// TwinCAT 3 PLC project CNM_OpModeHandlingInterfaces
// Title: CNM_OpModeHandlingInterfaces
// Company: ekvip automation GmbH
// Author: tsch
// ProjectVersion: 0.1.1.0
// Description: Providing interfaces that define handling operation modes in an industrial machine.
// ProgramVersion: 3.1.4026.19
// libraries:
//   CNM_AbstractObject, * (ekvip automation GmbH)
//   CNM_MessageInterfaces, * (ekvip automation GmbH)
//   CNM_ReturnTypes, * (ekvip automation GmbH)
//   Tc2_System, * (Beckhoff Automation GmbH)
// project tree:
//   Interfaces/Handler/ IOpModeHandlerMessageService.TcIO, INodeRequestProvider.TcIO, IOpModeHandler.TcIO, ISafetyReleaseDistributor.TcIO, ISafetySwitch.TcIO, IOpModeHandlerHmi.TcIO
//   Interfaces/Hmi/ IHmiApi.TcIO, IModeConditionProvider.TcIO
//   Interfaces/ IRunable.TcIO
//   Interfaces/Mode/ IModeBehaviour.TcIO, IModeProvider.TcIO, IModeSelect.TcIO
//   Interfaces/Node/Base/ INode.TcIO, INodeControl.TcIO, INodeRequest.TcIO
//   Interfaces/Node/ ICyclicNode.TcIO, INodeMessageService.TcIO
//   Interfaces/Node/OperationalNode/ IModeNode.TcIO, IOpModes.TcIO
//   Project Information/ F_GetCompany.TcPOU, F_GetTitle.TcPOU, F_GetVersion.TcPOU
//   Types/ ButtonStruct.TcDUT, HmiStates.TcDUT, ModeControlButtonStruct.TcDUT, NodeHandlerControlStruct.TcDUT
//   Version/ Global_Version.TcGVL

// ---- Types/ButtonStruct.TcDUT
TYPE ButtonStruct :
STRUCT
	text : Tc2_System.T_MaxString;
	enabled :BOOL := FALSE;
	visible :BOOL := FALSE;
	pressed :BOOL := FALSE;
END_STRUCT
END_TYPE

// ---- Types/HmiStates.TcDUT
{attribute 'qualified_only'}
{attribute 'strict'}
{attribute 'to_string'}
TYPE HmiStates :
(
	STOPPED := 0,
	HOME,
	RUNNING,
	PAUSE,
	STOP_PENDING,
	OFFLINE
);
END_TYPE

// ---- Types/ModeControlButtonStruct.TcDUT
TYPE ModeControlButtonStruct :
STRUCT
	Start :ButtonStruct:= (text:='%l%start%/l%');
	Stop :ButtonStruct:= (text:='%l%stop%/l%');
	StopRequest :ButtonStruct:= (text:='%l%stopRequest%/l%');
	StepMode :ButtonStruct:= (text:='%l%stepMode%/l%');
	Pause :ButtonStruct:= (text:='%l%pause%/l%');
END_STRUCT
END_TYPE

// ---- Types/NodeHandlerControlStruct.TcDUT
TYPE NodeHandlerControlStruct :
STRUCT
	stop :BOOL; // stop request for stop after end of cycle
	override :LREAL; // velocity orverride in % [0.0 ... 100.0]
END_STRUCT
END_TYPE

// ---- Version/Global_Version.TcGVL
{attribute 'TcGenerated'}
{attribute 'no-analysis'}
{attribute 'linkalways'}
// This function has been automatically generated from the project information.
VAR_GLOBAL CONSTANT
	{attribute 'const_non_replaced'}
	stLibVersion_CNM_OpModeHandlingInterfaces : ST_LibVersion := (iMajor := 0, iMinor := 1, iBuild := 1, iRevision := 0, nFlags := 0, sVersion := '0.1.1.0');
END_VAR

// ---- Interfaces/Handler/IOpModeHandlerMessageService.TcIO
(*
## short summary

This interface extends the IMessageInterface with the possibility to inject a global message service where the errors will be forwarded to.

legal notes
=================
| SPDX-FileCopyrightText: © 2024 ekvip automation GmbH <info@ekvip.de>
| SPDX-License-Identifier: Apache-2.0
| For details check: Apache-2.0_

.. _Apache-2.0: https://www.apache.org/licenses/LICENSE-2.0

.. </legal notes>  

*)

INTERFACE IOpModeHandlerMessageService EXTENDS CNM_MessageInterfaces.IMessageService

(*
## short summary

This property can be used to set the global message service interface during initialization.
The node message service will inform the node about the error and then forward the error to the global message service for handling the error.

legal notes
=================
| SPDX-FileCopyrightText: © 2025 ekvip automation GmbH <info@ekvip.de>
| SPDX-License-Identifier: Apache-2.0
| For details check: Apache-2.0_

.. _Apache-2.0: https://www.apache.org/licenses/LICENSE-2.0

.. </legal notes>  

*)

PROPERTY globalMessageService :CNM_MessageInterfaces.IMessageService
SET
END_SET
END_PROPERTY

END_INTERFACE

// ---- Interfaces/Handler/INodeRequestProvider.TcIO
(*
## short summary

This interface provides interfaces for the default node requests: disable, enable, initialize and stopImmediate.

legal notes
=================
| SPDX-FileCopyrightText: © 2024 ekvip automation GmbH <info@ekvip.de>
| SPDX-License-Identifier: Apache-2.0
| For details check: Apache-2.0_

.. _Apache-2.0: https://www.apache.org/licenses/LICENSE-2.0

.. </legal notes>  

*)

INTERFACE INodeRequestProvider EXTENDS __SYSTEM.IQueryInterface

(*
## short summary

This property returns the interface for the disabling request.

legal notes
=================
| SPDX-FileCopyrightText: © 2024 ekvip automation GmbH <info@ekvip.de>
| SPDX-License-Identifier: Apache-2.0
| For details check: Apache-2.0_

.. _Apache-2.0: https://www.apache.org/licenses/LICENSE-2.0

.. </legal notes>  

*)

PROPERTY disable :INodeRequest
GET
END_GET
END_PROPERTY

(*
## short summary

This property returns the interface for the disabling request.

legal notes
=================
| SPDX-FileCopyrightText: © 2024 ekvip automation GmbH <info@ekvip.de>
| SPDX-License-Identifier: Apache-2.0
| For details check: Apache-2.0_

.. _Apache-2.0: https://www.apache.org/licenses/LICENSE-2.0

.. </legal notes>  

*)

PROPERTY enable :INodeRequest
GET
END_GET
END_PROPERTY

(*
## short summary

This property returns the interface for the disabling request.

legal notes
=================
| SPDX-FileCopyrightText: © 2024 ekvip automation GmbH <info@ekvip.de>
| SPDX-License-Identifier: Apache-2.0
| For details check: Apache-2.0_

.. _Apache-2.0: https://www.apache.org/licenses/LICENSE-2.0

.. </legal notes>  

*)

PROPERTY initialize :INodeRequest
GET
END_GET
END_PROPERTY

(*
## short summary

This property returns the interface for the disabling request.

legal notes
=================
| SPDX-FileCopyrightText: © 2024 ekvip automation GmbH <info@ekvip.de>
| SPDX-License-Identifier: Apache-2.0
| For details check: Apache-2.0_

.. _Apache-2.0: https://www.apache.org/licenses/LICENSE-2.0

.. </legal notes>  

*)

PROPERTY stopImmediate :INodeRequest
GET
END_GET
END_PROPERTY

END_INTERFACE

// ---- Interfaces/Handler/IOpModeHandler.TcIO
(*
## short summary

This interface provides the cyclic run method and the fluent requests interface for a operation mode handler.

legal notes
=================
| SPDX-FileCopyrightText: © 2024 ekvip automation GmbH <info@ekvip.de>
| SPDX-License-Identifier: Apache-2.0
| For details check: Apache-2.0_

.. _Apache-2.0: https://www.apache.org/licenses/LICENSE-2.0

.. </legal notes>  

*)
INTERFACE IOpModeHandler EXTENDS CNM_AbstractObject.IObject, ISafetySwitch, IOpModeHandlerHmi, IRunable

END_INTERFACE

// ---- Interfaces/Handler/ISafetyReleaseDistributor.TcIO
(*
## short summary

This interface provides an subscription for a global safety release notification and should be implemented by the safety handler.

legal notes
=================
| SPDX-FileCopyrightText: © 2024 ekvip automation GmbH <info@ekvip.de>
| SPDX-License-Identifier: Apache-2.0
| For details check: Apache-2.0_

.. _Apache-2.0: https://www.apache.org/licenses/LICENSE-2.0

.. </legal notes>  

*)

INTERFACE ISafetyReleaseDistributor EXTENDS IRunable

(*
## short summary

This method adds the subscriber to a subscribption list. All subscribers are going to be notified, if the safety release changes.

legal notes
=================
| SPDX-FileCopyrightText: © 2022 ekvip automation GmbH <info@ekvip.de>
| SPDX-License-Identifier: Apache-2.0
| For details check: Apache-2.0_

.. _Apache-2.0: https://www.apache.org/licenses/LICENSE-2.0

.. </legal notes>  

*)

METHOD subscribe
VAR_INPUT
	(* class with the Interface ISafetySwitch, that can be switched on/off *)
	subscriber	:ISafetySwitch;
END_VAR
END_METHOD

END_INTERFACE

// ---- Interfaces/Handler/ISafetySwitch.TcIO
(*
## short summary

This interface needs to be implemented for a subscription to the ISafetyReleaseDistributer interface.
The provided methods switchOn and switchOff are automatically called if the safety release changes.

legal notes
=================
| SPDX-FileCopyrightText: © 2024 ekvip automation GmbH <info@ekvip.de>
| SPDX-License-Identifier: Apache-2.0
| For details check: Apache-2.0_

.. _Apache-2.0: https://www.apache.org/licenses/LICENSE-2.0

.. </legal notes>  

*)

INTERFACE ISafetySwitch EXTENDS CNM_AbstractObject.IObject

(*
## short summary

This property indicates that the unit is enabled and all safety requirements are met.

legal notes
=================
| SPDX-FileCopyrightText: © 2024 ekvip automation GmbH <info@ekvip.de>
| SPDX-License-Identifier: Apache-2.0
| For details check: Apache-2.0_

.. _Apache-2.0: https://www.apache.org/licenses/LICENSE-2.0

.. </legal notes>  

*)
PROPERTY isSwitchedOn : BOOL
GET
END_GET
END_PROPERTY

(*
## short summary

This method disables the unit if not all safety requirements are met. It Should be called only from the safety management.

legal notes
=================
| SPDX-FileCopyrightText: © 2024 ekvip automation GmbH <info@ekvip.de>
| SPDX-License-Identifier: Apache-2.0
| For details check: Apache-2.0_

.. _Apache-2.0: https://www.apache.org/licenses/LICENSE-2.0

.. </legal notes>  

*)

METHOD switchOff
END_METHOD

(*
## short summary

This method enables the unit if all safety requirements are met. It Should be called only from the safety management.

legal notes
=================
| SPDX-FileCopyrightText: © 2024 ekvip automation GmbH <info@ekvip.de>
| SPDX-License-Identifier: Apache-2.0
| For details check: Apache-2.0_

.. _Apache-2.0: https://www.apache.org/licenses/LICENSE-2.0

.. </legal notes>  

*)

METHOD switchOn
END_METHOD

END_INTERFACE

// ---- Interfaces/Handler/IOpModeHandlerHmi.TcIO
(*
## short summary
This interface provides an API to control the operation mode handler.

legal notes
=================
| SPDX-FileCopyrightText: © 2024 ekvip automation GmbH <info@ekvip.de>
| SPDX-License-Identifier: Apache-2.0
| For details check: Apache-2.0_

.. _Apache-2.0: https://www.apache.org/licenses/LICENSE-2.0

.. </legal notes>  

*)
INTERFACE IOpModeHandlerHmi EXTENDS CNM_AbstractObject.IObject

(*
## short summary
This methods enables the stepping operation on a given node and all of its subnodes.

legal notes
=================
| SPDX-FileCopyrightText: © 2025 ekvip automation GmbH <info@ekvip.de>
| SPDX-License-Identifier: Apache-2.0
| For details check: Apache-2.0_

.. _Apache-2.0: https://www.apache.org/licenses/LICENSE-2.0

.. </legal notes>  

*)

METHOD enableStepping : CNM_ReturnTypes.SingleExecutionResult
VAR_INPUT
	(* the node on which stepping should be enabled *)
	node :INode;
END_VAR
END_METHOD

(*
## short summary
This property can be used to inject a message service. Messages will be forwarded to that message service if it is set.

legal notes
=================
| SPDX-FileCopyrightText: © 2025 ekvip automation GmbH <info@ekvip.de>
| SPDX-License-Identifier: Apache-2.0
| For details check: Apache-2.0_

.. _Apache-2.0: https://www.apache.org/licenses/LICENSE-2.0

.. </legal notes>  

*)

PROPERTY globalMessageService : CNM_MessageInterfaces.IMessageService
SET
END_SET
END_PROPERTY

(*
## short summary
This property can be used to set the global override from the HMI and to read back the current override for the HMI.

**information**: the override has a range from 0.0 to 100.0 and will be limited to the upper/lower bound.

legal notes
=================
| SPDX-FileCopyrightText: © 2024 ekvip automation GmbH <info@ekvip.de>
| SPDX-License-Identifier: Apache-2.0
| For details check: Apache-2.0_

.. _Apache-2.0: https://www.apache.org/licenses/LICENSE-2.0

.. </legal notes>  

*)

PROPERTY globalOverride : LREAL
GET
END_GET
SET
END_SET
END_PROPERTY

(*
## short summary
This property indicates that a operation is being executed.

legal notes
=================
| SPDX-FileCopyrightText: © 2025 ekvip automation GmbH <info@ekvip.de>
| SPDX-License-Identifier: Apache-2.0
| For details check: Apache-2.0_

.. _Apache-2.0: https://www.apache.org/licenses/LICENSE-2.0

.. </legal notes>  

*)

PROPERTY modeIsExecuting : BOOL
GET
END_GET
END_PROPERTY

(*
## short summary
This property can be used to pause the currently running operation mode from the HMI and to read back if the mode is paused.

legal notes
=================
| SPDX-FileCopyrightText: © 2024 ekvip automation GmbH <info@ekvip.de>
| SPDX-License-Identifier: Apache-2.0
| For details check: Apache-2.0_

.. _Apache-2.0: https://www.apache.org/licenses/LICENSE-2.0

.. </legal notes>  

*)

PROPERTY pause : BOOL
GET
END_GET
SET
END_SET
END_PROPERTY

(*
## short summary
This property returns the INodeHmiApi interface of the root node from this opmode handler.

legal notes
=================
| SPDX-FileCopyrightText: © 2024 ekvip automation GmbH <info@ekvip.de>
| SPDX-License-Identifier: Apache-2.0
| For details check: Apache-2.0_

.. _Apache-2.0: https://www.apache.org/licenses/LICENSE-2.0

.. </legal notes>  

*)

PROPERTY rootNode :INode
GET
END_GET
END_PROPERTY

(*
## short summary
This method sets a mode for the rootnode or, if specified, for a single node and its subnodes.
It is only allowed to overwrite the mode if the rootNode or the specified node is not in busy state.

legal notes
=================
| SPDX-FileCopyrightText: © 2024 ekvip automation GmbH <info@ekvip.de>
| SPDX-License-Identifier: Apache-2.0
| For details check: Apache-2.0_

.. _Apache-2.0: https://www.apache.org/licenses/LICENSE-2.0

.. </legal notes>  

## example
set it for the whole machine:
```
myOpmodeHandler.setMode(
	mode := automaticMode
);
```

overwrite the mode of specified node:
```
myOpmodeHandler.setMode(
	mode := serviceMode,
	node := despensingUnit
);
```

*)
METHOD setMode : CNM_ReturnTypes.SingleExecutionResult
VAR_INPUT
	(* the mode instance that should be set *)
	mode : IModeBehaviour;
	(* optionally: a specified node in the tree that is not the subtree (if 0, the rootNode will be adressed) *)
	node : IModeNode := 0;
END_VAR
END_METHOD

(*
## short summary
This method starts the currently selected operation mode if all safety requirements are met.

legal notes
=================
| SPDX-FileCopyrightText: © 2024 ekvip automation GmbH <info@ekvip.de>
| SPDX-License-Identifier: Apache-2.0
| For details check: Apache-2.0_

.. _Apache-2.0: https://www.apache.org/licenses/LICENSE-2.0

.. </legal notes>  

## example
```
CASE step OF
	0:	// choose and set mode
		IF (handler.setMode(automaticMode) = SUCCESS ) THEN
			step := 1;
		END_IF
	1:	// start mode
		IF (handler.startMode() = SUCCESS) THEN
			step := 2;
		END_IF
	2: // stop mode if requested
		IF ( stopRequested ) THEN
			IF ( handler.stopMode() = SUCCESS ) THEN
				step := 0;
			END_IF
		END_IF
END_CASE
```

*)

METHOD startMode :CNM_ReturnTypes.SingleExecutionResult
VAR_INPUT
	(* optionally: a specified node in the tree that is not the subtree (if 0, the rootNode will be adressed) *)
	node : INode := 0;
END_VAR
END_METHOD

(*
## short summary
This method stops the currently running operation mode.
If the immediately flag is set, the current operation modewill be aborted and the machine will execute a fast stop.
If it is not set, the stop request flag for all nodes will be set and the operation modes should exit with a defined state.

legal notes
=================
| SPDX-FileCopyrightText: © 2024 ekvip automation GmbH <info@ekvip.de>
| SPDX-License-Identifier: Apache-2.0
| For details check: Apache-2.0_

.. _Apache-2.0: https://www.apache.org/licenses/LICENSE-2.0

.. </legal notes>  

## parameters
**return**: `CNM_ReturnTypes.SingleExecutionState`
- `SUCCESS`: the mode was stopped
- `BUSY`: mode is still stopping

## example
```
CASE step OF
	0:	// choose and set mode
		IF (handler.setMode(automaticMode) = SUCCESS ) THEN
			step := 1;
		END_IF
	1:	// start mode
		IF (handler.startMode() = SUCCESS) THEN
			step := 2;
		END_IF
	2: // stop mode if requested
		IF ( stopRequested ) THEN
			IF ( handler.stopMode() = SUCCESS ) THEN
				step := 0;
			END_IF
		END_IF
END_CASE
```

*)

METHOD stopMode : CNM_ReturnTypes.SingleExecutionState
VAR_INPUT
	(* if this flag is set, the current operation mode will be aborted and the machine will execute a fast stop *)
	immediately :BOOL := FALSE;
END_VAR
END_METHOD

END_INTERFACE

// ---- Interfaces/Hmi/IHmiApi.TcIO
(*
## short summary

This interface provides control methods and properties for a HMI handler class that are called by the CNM HMI framework.

legal notes
=================
| SPDX-FileCopyrightText: © 2024 ekvip automation GmbH <info@ekvip.de>
| SPDX-License-Identifier: Apache-2.0
| For details check: Apache-2.0_

.. _Apache-2.0: https://www.apache.org/licenses/LICENSE-2.0

.. </legal notes>  

*)

INTERFACE IHmiApi EXTENDS __SYSTEM.IQueryInterface, IRunable

(*
## short summary

This method returns the instance path of the root node of the operation mode handler.
It is used for the HMI tree building mechanism.

legal notes
=================
| SPDX-FileCopyrightText: © 2024 ekvip automation GmbH <info@ekvip.de>
| SPDX-License-Identifier: Apache-2.0
| For details check: Apache-2.0_

.. _Apache-2.0: https://www.apache.org/licenses/LICENSE-2.0

.. </legal notes>  

*)

{attribute 'TcRpcEnable'}
METHOD getRootNodeName : Tc2_System.T_MaxString
END_METHOD

(*
## short summary

This property is true if the operation mode handler has a safety release.

legal notes
=================
| SPDX-FileCopyrightText: © 2024 ekvip automation GmbH <info@ekvip.de>
| SPDX-License-Identifier: Apache-2.0
| For details check: Apache-2.0_

.. _Apache-2.0: https://www.apache.org/licenses/LICENSE-2.0

.. </legal notes>  

*)

{attribute 'monitoring':='call'}
PROPERTY IsSafetyOk : BOOL
GET
END_GET
END_PROPERTY

(*
## short summary

This property can returns the root node state for currently active operation mode.

legal notes
=================
| SPDX-FileCopyrightText: © 2024 ekvip automation GmbH <info@ekvip.de>
| SPDX-License-Identifier: Apache-2.0
| For details check: Apache-2.0_

.. _Apache-2.0: https://www.apache.org/licenses/LICENSE-2.0

.. </legal notes>  

*)

{attribute 'monitoring' := 'call'}
PROPERTY OpModeState : CNM_ReturnTypes.SingleExecutionState
GET
END_GET
END_PROPERTY

(*
## short summary

This property can be used to pause the currently running operation mode from the HMI and to read back if the mode is paused.

legal notes
=================
| SPDX-FileCopyrightText: © 2024 ekvip automation GmbH <info@ekvip.de>
| SPDX-License-Identifier: Apache-2.0
| For details check: Apache-2.0_

.. _Apache-2.0: https://www.apache.org/licenses/LICENSE-2.0

.. </legal notes>  

*)

{attribute 'monitoring':='call'}
PROPERTY pause : BOOL
GET
END_GET
SET
END_SET
END_PROPERTY

(*
## short summary

This property shows that the root node (and so the whole machine) is waiting for a step signal when step mode is enabled.

legal notes
=================
| SPDX-FileCopyrightText: © 2024 ekvip automation GmbH <info@ekvip.de>
| SPDX-License-Identifier: Apache-2.0
| For details check: Apache-2.0_

.. _Apache-2.0: https://www.apache.org/licenses/LICENSE-2.0

.. </legal notes>  

*)

{attribute 'monitoring' := 'call'}
PROPERTY rootNodeWaitingForStep : BOOL
GET
END_GET
END_PROPERTY

(*
## short summary

This property setter sends the step signal to all nodes of the machine.
If the step mode is enabled, the step signal will be set for exactly one PLC cycle.
If the step mode isn't enabled, the step signal won't have any effect at all.

legal notes
=================
| SPDX-FileCopyrightText: © 2024 ekvip automation GmbH <info@ekvip.de>
| SPDX-License-Identifier: Apache-2.0
| For details check: Apache-2.0_

.. _Apache-2.0: https://www.apache.org/licenses/LICENSE-2.0

.. </legal notes>  

*)

{attribute 'monitoring':='call'}
PROPERTY step : BOOL
SET
END_SET
END_PROPERTY

END_INTERFACE

// ---- Interfaces/Hmi/IModeConditionProvider.TcIO
(*
## short summary

This interface provides a method that checks for each mode if it can be started.

legal notes
=================
| SPDX-FileCopyrightText: © 2024 ekvip automation GmbH <info@ekvip.de>
| SPDX-License-Identifier: Apache-2.0
| For details check: Apache-2.0_

.. _Apache-2.0: https://www.apache.org/licenses/LICENSE-2.0

.. </legal notes>  

*)

INTERFACE IModeConditionProvider

(*
## short summary

This method checks the start conditions for the selected operation mode.
If the mode is allowed to be started, it returns TRUE.

legal notes
=================
| SPDX-FileCopyrightText: © 2024 ekvip automation GmbH <info@ekvip.de>
| SPDX-License-Identifier: Apache-2.0
| For details check: Apache-2.0_

.. _Apache-2.0: https://www.apache.org/licenses/LICENSE-2.0

.. </legal notes>  

*)

METHOD checkModeIsAllowed : BOOL
VAR_INPUT
	mode :UDINT;
	node :INode;
END_VAR
END_METHOD

END_INTERFACE

// ---- Interfaces/IRunable.TcIO
(*
## short summary

This interface provides a void run() method without parameters.

legal notes
=================
| SPDX-FileCopyrightText: © 2025 ekvip automation GmbH <info@ekvip.de>
| SPDX-License-Identifier: Apache-2.0
| For details check: Apache-2.0_

.. _Apache-2.0: https://www.apache.org/licenses/LICENSE-2.0

.. </legal notes>  

*)

INTERFACE IRunable EXTENDS CNM_AbstractObject.IObject

(*
## short summary

A method that should be called cyclically to update and execute a class instance.

legal notes
=================
| SPDX-FileCopyrightText: © 2025 ekvip automation GmbH <info@ekvip.de>
| SPDX-License-Identifier: Apache-2.0
| For details check: Apache-2.0_

.. _Apache-2.0: https://www.apache.org/licenses/LICENSE-2.0

.. </legal notes>  

*)

METHOD run
END_METHOD

END_INTERFACE

// ---- Interfaces/Mode/IModeBehaviour.TcIO
(*
## short summary

This interface defines the methods needed for the mode delegates.

legal notes
=================
| SPDX-FileCopyrightText: © 2024 ekvip automation GmbH <info@ekvip.de>
| SPDX-License-Identifier: Apache-2.0
| For details check: Apache-2.0_

.. _Apache-2.0: https://www.apache.org/licenses/LICENSE-2.0

.. </legal notes>  

*)

INTERFACE IModeBehaviour EXTENDS CNM_AbstractObject.IObject

(*
## short summary

This property is intended to inform cyclic nodes (devices) that manual commands are allowed to be executed.
Usually only the manual mode behaviour sets this to true, but it may be also used for other custom modes if needed.

legal notes
=================
| SPDX-FileCopyrightText: © 2024 ekvip automation GmbH <info@ekvip.de>
| SPDX-License-Identifier: Apache-2.0
| For details check: Apache-2.0_

.. _Apache-2.0: https://www.apache.org/licenses/LICENSE-2.0

.. </legal notes>  

*)

PROPERTY enableManCmds : BOOL
GET
END_GET
END_PROPERTY

(*
## short summary

This method is called once for every node when a new oepration mode is started.
It is intended to inform the node that a new mode is startet, so you can throw events / MES notifications /  do data management here.

legal notes
=================
| SPDX-FileCopyrightText: © 2024 ekvip automation GmbH <info@ekvip.de>
| SPDX-License-Identifier: Apache-2.0
| For details check: Apache-2.0_

.. _Apache-2.0: https://www.apache.org/licenses/LICENSE-2.0

.. </legal notes>  

*)

METHOD enterMode
VAR_INPUT
	node : IOpModes;
END_VAR
END_METHOD

(*
## short summary

This method is called once for every node when the current operation mode is stopped.
It is intended to inform the node that the mode is stopped, so you can throw events / MES notifications /  do data management here.

legal notes
=================
| SPDX-FileCopyrightText: © 2024 ekvip automation GmbH <info@ekvip.de>
| SPDX-License-Identifier: Apache-2.0
| For details check: Apache-2.0_

.. _Apache-2.0: https://www.apache.org/licenses/LICENSE-2.0

.. </legal notes>  

*)

METHOD exitMode
VAR_INPUT
	node : IOpModes;
END_VAR
END_METHOD

(*
## short summary

This property returns the id that was used to request the mode delegate.
The mode provider class has to set it.

legal notes
=================
| SPDX-FileCopyrightText: © 2024 ekvip automation GmbH <info@ekvip.de>
| SPDX-License-Identifier: Apache-2.0
| For details check: Apache-2.0_

.. _Apache-2.0: https://www.apache.org/licenses/LICENSE-2.0

.. </legal notes>  

*)

PROPERTY id : UDINT
GET
END_GET
SET
END_SET
END_PROPERTY

(*
## short summary

This method is calling the operation mode methods for every node depending on the current behaviour.

legal notes
=================
| SPDX-FileCopyrightText: © 2024 ekvip automation GmbH <info@ekvip.de>
| SPDX-License-Identifier: Apache-2.0
| For details check: Apache-2.0_

.. _Apache-2.0: https://www.apache.org/licenses/LICENSE-2.0

.. </legal notes>  

*)

METHOD run :CNM_ReturnTypes.SingleExecutionState
VAR_INPUT
	execute :BOOL;
	pause :BOOL;
	node :IOpModes;
END_VAR
END_METHOD

END_INTERFACE

// ---- Interfaces/Mode/IModeProvider.TcIO
(*
## short summary

This interface defines method for a mode behaviour provider. 
It can be used to inject custom modes into the HMI class.  

legal notes
=================
| SPDX-FileCopyrightText: © 2024 ekvip automation GmbH <info@ekvip.de>
| SPDX-License-Identifier: Apache-2.0
| For details check: Apache-2.0_

.. _Apache-2.0: https://www.apache.org/licenses/LICENSE-2.0

.. </legal notes>  

*)

INTERFACE IModeProvider EXTENDS CNM_AbstractObject.IObject

(*
## short summary

A method that returns an interface to an instance of a mode behaviour.
It can be used to trabnslate the operation mode enum to a mode delegate. Overwrite this method for custom modes.

legal notes
=================
| SPDX-FileCopyrightText: © 2024 ekvip automation GmbH <info@ekvip.de>
| SPDX-License-Identifier: Apache-2.0
| For details check: Apache-2.0_

.. _Apache-2.0: https://www.apache.org/licenses/LICENSE-2.0

.. </legal notes>  

*)

METHOD getMode : IModeBehaviour
VAR_INPUT
	mode :UDINT;
END_VAR
END_METHOD

(*
## short summary

This property returns an IModeSelect that offers properties for the mandatory modes.
The modes are accessable via fluent interface, e.g. myModeFactory.mode.automaticMode.

legal notes
=================
| SPDX-FileCopyrightText: © 2024 ekvip automation GmbH <info@ekvip.de>
| SPDX-License-Identifier: Apache-2.0
| For details check: Apache-2.0_

.. _Apache-2.0: https://www.apache.org/licenses/LICENSE-2.0

.. </legal notes>  

*)

PROPERTY mode : IModeSelect
GET
END_GET
END_PROPERTY

END_INTERFACE

// ---- Interfaces/Mode/IModeSelect.TcIO
(*
## short summary

This is an interface to fluently provide the mandatory mode behaviours.

legal notes
=================
| SPDX-FileCopyrightText: © 2024 ekvip automation GmbH <info@ekvip.de>
| SPDX-License-Identifier: Apache-2.0
| For details check: Apache-2.0_

.. _Apache-2.0: https://www.apache.org/licenses/LICENSE-2.0

.. </legal notes>  

*)

INTERFACE IModeSelect EXTENDS CNM_AbstractObject.IObject

(*
## short summary

This property returns an IModeBehaviour that implements the delegate for the automatic mode.

legal notes
=================
| SPDX-FileCopyrightText: © 2024 ekvip automation GmbH <info@ekvip.de>
| SPDX-License-Identifier: Apache-2.0
| For details check: Apache-2.0_

.. _Apache-2.0: https://www.apache.org/licenses/LICENSE-2.0

.. </legal notes>  

*)
PROPERTY automaticMode : IModeBehaviour
GET
END_GET
END_PROPERTY

(*
## short summary

This property returns an IModeBehaviour that implements the delegate for the homing mode.

legal notes
=================
| SPDX-FileCopyrightText: © 2024 ekvip automation GmbH <info@ekvip.de>
| SPDX-License-Identifier: Apache-2.0
| For details check: Apache-2.0_

.. _Apache-2.0: https://www.apache.org/licenses/LICENSE-2.0

.. </legal notes>  

*)

PROPERTY homingMode : IModeBehaviour
GET
END_GET
END_PROPERTY

(*
## short summary

This property returns an IModeBehaviour that implements the delegate for the manual mode.

legal notes
=================
| SPDX-FileCopyrightText: © 2024 ekvip automation GmbH <info@ekvip.de>
| SPDX-License-Identifier: Apache-2.0
| For details check: Apache-2.0_

.. _Apache-2.0: https://www.apache.org/licenses/LICENSE-2.0

.. </legal notes>  

*)

PROPERTY manualMode : IModeBehaviour
GET
END_GET
END_PROPERTY

(*
## short summary

This property returns an IModeBehaviour that implements the delegate for no operation mode.

legal notes
=================
| SPDX-FileCopyrightText: © 2025 ekvip automation GmbH <info@ekvip.de>
| SPDX-License-Identifier: Apache-2.0
| For details check: Apache-2.0_

.. _Apache-2.0: https://www.apache.org/licenses/LICENSE-2.0

.. </legal notes>  

*)

PROPERTY noMode : IModeBehaviour
GET
END_GET
END_PROPERTY

END_INTERFACE

// ---- Interfaces/Node/Base/INode.TcIO
(*
## short summary
This interface provides methods and properties that every node needs to implement.
Some of the methods and properties are used for the CNM HMI framework.

legal notes
=================
| SPDX-FileCopyrightText: © 2024 ekvip automation GmbH <info@ekvip.de>
| SPDX-License-Identifier: Apache-2.0
| For details check: Apache-2.0_

.. _Apache-2.0: https://www.apache.org/licenses/LICENSE-2.0

.. </legal notes>  

*)

INTERFACE INode EXTENDS CNM_AbstractObject.IObject

(*
## short summary
This property returns the id of the mode that is currently propagated.
It reflects the hmi selection.

legal notes
=================
| SPDX-FileCopyrightText: © 2024 ekvip automation GmbH <info@ekvip.de>
| SPDX-License-Identifier: Apache-2.0
| For details check: Apache-2.0_

.. _Apache-2.0: https://www.apache.org/licenses/LICENSE-2.0

.. </legal notes>  

*)

PROPERTY currentModeId : UDINT
GET
END_GET
END_PROPERTY

(*
## short summary
This method disables a node (E.g. axes should be disabled). It can take mutliple cycles. It has to be implemented for every node/device.
The execute input needs a rising edge to execute the method.
If there is nothing to disable, just return a 'SUCCESS' state.

This method is called automatically by the operation mode handler.

legal notes
=================
| SPDX-FileCopyrightText: © 2024 ekvip automation GmbH <info@ekvip.de>
| SPDX-License-Identifier: Apache-2.0
| For details check: Apache-2.0_

.. _Apache-2.0: https://www.apache.org/licenses/LICENSE-2.0

.. </legal notes>  

*)

METHOD disable : CNM_ReturnTypes.SingleExecutionState
VAR_INPUT
	execute :BOOL;
END_VAR
END_METHOD

(*
## short summary
This method enables a node. It can take mutliple cycles. It has to be implemented for every node/device.
The intention is to enable devices here, e.g. axes, laser, dispenser etc.
The execute input needs a rising edge to execute the method.
If there is nothing to enable, just return a 'SUCCESS' state.

This method is called automatically by the operation mode handler.

legal notes
=================
| SPDX-FileCopyrightText: © 2024 ekvip automation GmbH <info@ekvip.de>
| SPDX-License-Identifier: Apache-2.0
| For details check: Apache-2.0_

.. _Apache-2.0: https://www.apache.org/licenses/LICENSE-2.0

.. </legal notes>  

*)
METHOD enable : CNM_ReturnTypes.SingleExecutionState
VAR_INPUT
	execute :BOOL;
END_VAR
END_METHOD

(*
## short summary
This property is used to enable/disable manual stepping.

legal notes
=================
| SPDX-FileCopyrightText: © 2025 ekvip automation GmbH <info@ekvip.de>
| SPDX-License-Identifier: Apache-2.0
| For details check: Apache-2.0_

.. _Apache-2.0: https://www.apache.org/licenses/LICENSE-2.0

.. </legal notes>  

*)

PROPERTY enableStepping : BOOL
GET
END_GET
SET
END_SET
END_PROPERTY

(*
## short summary
This method returns the variable name for a subnode at a given array index of the internal array list.
It is required for the HMI connection to construct the node tree from the PLC on HMI side.
It is also intended to be called from the HMI via remote procedure call.

legal notes
=================
| SPDX-FileCopyrightText: © 2024 ekvip automation GmbH <info@ekvip.de>
| SPDX-License-Identifier: Apache-2.0
| For details check: Apache-2.0_

.. _Apache-2.0: https://www.apache.org/licenses/LICENSE-2.0

.. </legal notes>  

*)

METHOD getSubnodeName : CNM_AbstractObject.ObjectName
VAR_INPUT
	(*  index of a subnode in the subnode array list *)
	index :UDINT;
END_VAR
END_METHOD

(*
## short summary
This property indicates whether a node has an error. It is used by the CNM HMI.

legal notes
=================
| SPDX-FileCopyrightText: © 2024 ekvip automation GmbH <info@ekvip.de>
| SPDX-License-Identifier: Apache-2.0
| For details check: Apache-2.0_

.. _Apache-2.0: https://www.apache.org/licenses/LICENSE-2.0

.. </legal notes>  

*)
{attribute 'monitoring' := 'call'}
PROPERTY hasError : BOOL
GET
END_GET
SET
END_SET
END_PROPERTY

(*
## short summary
This method contains instructions and sequences for the init mode.
This mode is intended for initializing a machine, e.g. set references and parameters, establish a connection to global production systems (MES).
If the node should do nothing, return a 'SUCCESS'.
It should run until all initializations are done or the mode is stopped immedtiately or a stop request is raised.
This method is called automatically by the operation mode handler after PLC startup.

legal notes
=================
| SPDX-FileCopyrightText: © 2024 ekvip automation GmbH <info@ekvip.de>
| SPDX-License-Identifier: Apache-2.0
| For details check: Apache-2.0_

.. _Apache-2.0: https://www.apache.org/licenses/LICENSE-2.0

.. </legal notes>  

*)
METHOD initialize : CNM_ReturnTypes.SingleExecutionState
VAR_INPUT
	execute :BOOL;
END_VAR
END_METHOD

(*
## short summary
This property indicates that a node or subunit is home position. The getter evaluates the home property of all child nodes.  
It is used by the CNM HMI.

legal notes
=================
| SPDX-FileCopyrightText: © 2024 ekvip automation GmbH <info@ekvip.de>
| SPDX-License-Identifier: Apache-2.0
| For details check: Apache-2.0_

.. _Apache-2.0: https://www.apache.org/licenses/LICENSE-2.0

.. </legal notes>  

*)
{attribute 'monitoring' := 'call'}
PROPERTY isInHome : BOOL
GET
END_GET
SET
END_SET
END_PROPERTY

(*
## short summary
This property indicates that a node or subunit is waiting for a step signal. It is used by the CNM HMI.

legal notes
=================
| SPDX-FileCopyrightText: © 2024 ekvip automation GmbH <info@ekvip.de>
| SPDX-License-Identifier: Apache-2.0
| For details check: Apache-2.0_

.. _Apache-2.0: https://www.apache.org/licenses/LICENSE-2.0

.. </legal notes>  

*)
{attribute 'monitoring' := 'call'}
PROPERTY isWaitingForStep : BOOL
GET
END_GET
SET
END_SET
END_PROPERTY

(*
## short summary
This property is used to set a local override for single node. 
The local override will be multiplied with the global override.

legal notes
=================
| SPDX-FileCopyrightText: © 2024 ekvip automation GmbH <info@ekvip.de>
| SPDX-License-Identifier: Apache-2.0
| For details check: Apache-2.0_

.. _Apache-2.0: https://www.apache.org/licenses/LICENSE-2.0

.. </legal notes>  

*)
{attribute 'monitoring' := 'variable'}
PROPERTY localOverride : LREAL
GET
END_GET
SET
END_SET
END_PROPERTY

(*
## short summary
This property returns the interface to the instance mode data dto.

legal notes
=================
| SPDX-FileCopyrightText: © 2024 ekvip automation GmbH <info@ekvip.de>
| SPDX-License-Identifier: Apache-2.0
| For details check: Apache-2.0_

.. _Apache-2.0: https://www.apache.org/licenses/LICENSE-2.0

.. </legal notes>  

*)
PROPERTY nodeControl : INodeControl
GET
END_GET
END_PROPERTY

(*
## short summary
This property returns the state of the node for the current node request.
The unit is still running if the state is ''BUSY''.

legal notes
=================
| SPDX-FileCopyrightText: © 2024 ekvip automation GmbH <info@ekvip.de>
| SPDX-License-Identifier: Apache-2.0
| For details check: Apache-2.0_

.. _Apache-2.0: https://www.apache.org/licenses/LICENSE-2.0

.. </legal notes>  

*)
{attribute 'monitoring' := 'call'}
PROPERTY nodeState : CNM_ReturnTypes.SingleExecutionState
GET
END_GET
END_PROPERTY

(*
## short summary
This boolean can be used to set the step signal for a node for one plc cycle.

legal notes
=================
| SPDX-FileCopyrightText: © 2025 ekvip automation GmbH <info@ekvip.de>
| SPDX-License-Identifier: Apache-2.0
| For details check: Apache-2.0_

.. _Apache-2.0: https://www.apache.org/licenses/LICENSE-2.0

.. </legal notes>  

*)

PROPERTY step : BOOL
GET
END_GET
SET
END_SET
END_PROPERTY

(*
## short summary
This method executes stops all movements of a node. It has to be overwritten for every node.
E.g. axes should perform a quickstop, cylinders should be turned off, etc.
If the node should do nothing, return a 'SUCCESS'.
It should stop axes/cylinders/process (e.g. laser welding, dispensing) endless until the manual mode is stopped via stop request or immediate stop.
This method is called automatically by the operation mode handler before disabling the machine or if the operator selects an immediate stop.

**attention**: If this method returns the state 'ERROR', the operation mode handler automatically disables the whole machine!

legal notes
=================
| SPDX-FileCopyrightText: © 2024 ekvip automation GmbH <info@ekvip.de>
| SPDX-License-Identifier: Apache-2.0
| For details check: Apache-2.0_

.. _Apache-2.0: https://www.apache.org/licenses/LICENSE-2.0

.. </legal notes>  

*)

METHOD stopImmediate : CNM_ReturnTypes.SingleExecutionState
VAR_INPUT
	execute :BOOL;
END_VAR
END_METHOD

END_INTERFACE

// ---- Interfaces/Node/Base/INodeControl.TcIO
(*
## short summary

This interface provides a fluent way to access the global control signals (stopRequests, overrides, step requests).

legal notes
=================
| SPDX-FileCopyrightText: © 2024 ekvip automation GmbH <info@ekvip.de>
| SPDX-License-Identifier: Apache-2.0
| For details check: Apache-2.0_

.. _Apache-2.0: https://www.apache.org/licenses/LICENSE-2.0

.. </legal notes>  

*)
INTERFACE INodeControl EXTENDS __SYSTEM.IQueryInterface

(*
## short summary

This property returns the effective override for a node, which is the result of the multiplication of global and local override.

legal notes
=================
| SPDX-FileCopyrightText: © 2024 ekvip automation GmbH <info@ekvip.de>
| SPDX-License-Identifier: Apache-2.0
| For details check: Apache-2.0_

.. _Apache-2.0: https://www.apache.org/licenses/LICENSE-2.0

.. </legal notes>  

*)
PROPERTY override : LREAL
GET
END_GET
END_PROPERTY

(*
## short summary

This property represents the stop request signal which either the operator triggers from the HMI or which is set by an error.

legal notes
=================
| SPDX-FileCopyrightText: © 2024 ekvip automation GmbH <info@ekvip.de>
| SPDX-License-Identifier: Apache-2.0
| For details check: Apache-2.0_

.. _Apache-2.0: https://www.apache.org/licenses/LICENSE-2.0

.. </legal notes>  

*)
PROPERTY stopRequest : BOOL
GET
END_GET
END_PROPERTY

END_INTERFACE

// ---- Interfaces/Node/Base/INodeRequest.TcIO
(*
## short summary

This interface defines the methods needed for the node request delegates.

legal notes
=================
| SPDX-FileCopyrightText: © 2024 ekvip automation GmbH <info@ekvip.de>
| SPDX-License-Identifier: Apache-2.0
| For details check: Apache-2.0_

.. _Apache-2.0: https://www.apache.org/licenses/LICENSE-2.0

.. </legal notes>  

*)

INTERFACE INodeRequest EXTENDS __SYSTEM.IQueryInterface

(*
## short summary

This method is calling the node request methods for every node depending on the current request.

legal notes
=================
| SPDX-FileCopyrightText: © 2024 ekvip automation GmbH <info@ekvip.de>
| SPDX-License-Identifier: Apache-2.0
| For details check: Apache-2.0_

.. _Apache-2.0: https://www.apache.org/licenses/LICENSE-2.0

.. </legal notes>  

*)

METHOD run :CNM_ReturnTypes.SingleExecutionState
VAR_INPUT
	execute :BOOL;
	node :INode;
END_VAR
END_METHOD

END_INTERFACE

// ---- Interfaces/Node/ICyclicNode.TcIO
(*
## short summary

This interface extends the INode interface with a run method for a cyclically update/monitoring.
Examples for cyclic nodes are device drivers, meausurements or communication nodes (MES / other PLC / etc.)

legal notes
=================
| SPDX-FileCopyrightText: © 2024 ekvip automation GmbH <info@ekvip.de>
| SPDX-License-Identifier: Apache-2.0
| For details check: Apache-2.0_

.. _Apache-2.0: https://www.apache.org/licenses/LICENSE-2.0

.. </legal notes>  

*)

INTERFACE ICyclicNode EXTENDS INode

(*
## short summary

This method will be called in every cycle for a node. It can be used to implement hardware drivers/measurements/monitoring.
The returned state defines the overall state of the node. It should return BUSY when the node executes a command, otherwise SUCCESS( or IDLE if there is nothing to do).
(Simple monitoring is not a command an should return SUCCESS).

**attention**: the returned SingleExecutionState will be evaluated cyclically wihtin the node tree.
In case a node returns an ERROR state, the whole machine will be disabled.
Return ERROR only for fatal or critical errors and handle other errors within the node.

legal notes
=================
| SPDX-FileCopyrightText: © 2025 ekvip automation GmbH <info@ekvip.de>
| SPDX-License-Identifier: Apache-2.0
| For details check: Apache-2.0_

.. _Apache-2.0: https://www.apache.org/licenses/LICENSE-2.0

.. </legal notes>  

*)

METHOD run : CNM_ReturnTypes.SingleExecutionState
END_METHOD

END_INTERFACE

// ---- Interfaces/Node/INodeMessageService.TcIO
(*
## short summary

This interface extends the IMessageInterface with the possibility to inject a global message service where the errors will be forwarded to.

legal notes
=================
| SPDX-FileCopyrightText: © 2024 ekvip automation GmbH <info@ekvip.de>
| SPDX-License-Identifier: Apache-2.0
| For details check: Apache-2.0_

.. _Apache-2.0: https://www.apache.org/licenses/LICENSE-2.0

.. </legal notes>  

*)

INTERFACE INodeMessageService EXTENDS CNM_MessageInterfaces.IMessageService

(*
## short summary

This property can be used to set the global message service interface during initialization.
The node message service will inform the node about the error and then forward the error to the global message service for handling the error.

legal notes
=================
| SPDX-FileCopyrightText: © 2025 ekvip automation GmbH <info@ekvip.de>
| SPDX-License-Identifier: Apache-2.0
| For details check: Apache-2.0_

.. _Apache-2.0: https://www.apache.org/licenses/LICENSE-2.0

.. </legal notes>  

*)

PROPERTY globalMessageService : CNM_MessageInterfaces.IMessageService
SET
END_SET
END_PROPERTY

END_INTERFACE

// ---- Interfaces/Node/OperationalNode/IModeNode.TcIO
(*
## short summary
This interface defines the methods needed for operation mode dependent nodes.

legal notes
=================
| SPDX-FileCopyrightText: © 2024 ekvip automation GmbH <info@ekvip.de>
| SPDX-License-Identifier: Apache-2.0
| For details check: Apache-2.0_

.. _Apache-2.0: https://www.apache.org/licenses/LICENSE-2.0

.. </legal notes>  

*)

INTERFACE IModeNode EXTENDS INode, IOpModes

(*
## short summary
This property indicates that a node or subunit is empty (no parts are physically present). It is used for the HMI connection.

legal notes
=================
| SPDX-FileCopyrightText: © 2024 ekvip automation GmbH <info@ekvip.de>
| SPDX-License-Identifier: Apache-2.0
| For details check: Apache-2.0_

.. _Apache-2.0: https://www.apache.org/licenses/LICENSE-2.0

.. </legal notes>  

*)
{attribute 'monitoring' := 'call'}
PROPERTY isEmpty : BOOL
GET
END_GET
SET
END_SET
END_PROPERTY

(*
## short summary
This method allows the overwrite of the current mode state with a new mode, provided the current mode state is in `IDLE` or `SUCCESS` status,
and the input mode object is valid. It determines the outcome of the overwrite operation and returns the appropriate result.

legal notes
=================
| SPDX-FileCopyrightText: © 2024 ekvip automation GmbH <info@ekvip.de>
| SPDX-License-Identifier: Apache-2.0
| For details check: Apache-2.0_

.. _Apache-2.0: https://www.apache.org/licenses/LICENSE-2.0

.. </legal notes>  

## example

```
IF (opModeHandler.setMode(mode := automaticMode) = SingleExecutionResult.SUCCESS)
	AND_THEN (dispensingStation.overwriteMode(mode := simulatedMode) = SingleExecutionResult.SUCCESS)
THEN
	opModeHandler.startMode();
END_IF
```

*)
METHOD overwriteMode : CNM_ReturnTypes.SingleExecutionResult
VAR_INPUT
	mode : IModeBehaviour;
END_VAR
END_METHOD

(*
## short summary
This boolean can be used to set the step signal for a node for one plc cycle.

legal notes
=================
| SPDX-FileCopyrightText: © 2025 ekvip automation GmbH <info@ekvip.de>
| SPDX-License-Identifier: Apache-2.0
| For details check: Apache-2.0_

.. _Apache-2.0: https://www.apache.org/licenses/LICENSE-2.0

.. </legal notes>  

*)

PROPERTY step : BOOL
GET
END_GET
SET
END_SET
END_PROPERTY

END_INTERFACE

// ---- Interfaces/Node/OperationalNode/IOpModes.TcIO
(*
## short summary
This interface defines the methods needed for the mode delegates. Mandatory mode methods must be implemented for all nodes.

legal notes
=================
| SPDX-FileCopyrightText: © 2024 ekvip automation GmbH <info@ekvip.de>
| SPDX-License-Identifier: Apache-2.0
| For details check: Apache-2.0_

.. _Apache-2.0: https://www.apache.org/licenses/LICENSE-2.0

.. </legal notes>  

*)

INTERFACE IOpModes EXTENDS __SYSTEM.IQueryInterface

(*
## short summary
This method will be called once before a new mode is started. The method is called for exactly one cycle and
is therefore suitable for triggering events or sending messages to MES systems.
If the node should do nothing when changing the mode, leave it empty.

legal notes
=================
| SPDX-FileCopyrightText: © 2024 ekvip automation GmbH <info@ekvip.de>
| SPDX-License-Identifier: Apache-2.0
| For details check: Apache-2.0_

.. _Apache-2.0: https://www.apache.org/licenses/LICENSE-2.0

.. </legal notes>  

*)
METHOD enterNewMode
END_METHOD

(*
## short summary
This method will be called once after a mdoe was finished (stopped). The method is called for exactly one cycle and
is therefore suitable for triggering events or sending messages to MES systems.
If the node should do nothing when changing the mode, leave it empty.

legal notes
=================
| SPDX-FileCopyrightText: © 2024 ekvip automation GmbH <info@ekvip.de>
| SPDX-License-Identifier: Apache-2.0
| For details check: Apache-2.0_

.. _Apache-2.0: https://www.apache.org/licenses/LICENSE-2.0

.. </legal notes>  

*)
METHOD exitCurrentMode
END_METHOD

(*
## short summary
This method contains instructions and sequences for the automatic mode. It has to be overwritten for every node.
If the node should do nothing, return a 'SUCCESS'.
It should run in an endless loop until the mode is stopped immedtiately or a stop request is raised (THIS^.modeControl.stopRequest).
This method is called automatically by the operation mode handler.

**attention**: If this method returns the state 'ERROR', the operation mode handler automatically disables the whole machine!

legal notes
=================
| SPDX-FileCopyrightText: © 2024 ekvip automation GmbH <info@ekvip.de>
| SPDX-License-Identifier: Apache-2.0
| For details check: Apache-2.0_

.. _Apache-2.0: https://www.apache.org/licenses/LICENSE-2.0

.. </legal notes>  

*)
METHOD runAutomatic : CNM_ReturnTypes.SingleExecutionState
VAR_INPUT
	execute :BOOL;
	pause :BOOL;
END_VAR
END_METHOD

(*
## short summary
This method contains instructions and sequences for product type/variant changeover.
This mode is intended for loading recipe data and / or change type/variant specific production tools.
If the node should do nothing, return a 'SUCCESS'. If the changeove is finished, return 'SUCCESS'.

This method is called automatically by the operation mode handler.

**attention**: If this method returns the state 'ERROR', the operation mode handler automatically disables the whole machine!

legal notes
=================
| SPDX-FileCopyrightText: © 2025 ekvip automation GmbH <info@ekvip.de>
| SPDX-License-Identifier: Apache-2.0
| For details check: Apache-2.0_

.. _Apache-2.0: https://www.apache.org/licenses/LICENSE-2.0

.. </legal notes>  

*)

METHOD runChangeOver : CNM_ReturnTypes.SingleExecutionState
VAR_INPUT
	execute :BOOL;
	pause :BOOL;
END_VAR
END_METHOD

(*
## short summary
This method contains instructions and sequences for the clean up mode.
This mode is intended for running a machine empty and then cleaning up internal data.
If the node should do nothing, return a 'SUCCESS'.
It should run in an endless loop until the machine is empty or the mode is stopped immedtiately or a stop request is raised (THIS^.modeControl.stopRequest).
This method is called automatically by the operation mode handler.

**attention**: If this method returns the state 'ERROR', the operation mode handler automatically disables the whole machine!

legal notes
=================
| SPDX-FileCopyrightText: © 2024 ekvip automation GmbH <info@ekvip.de>
| SPDX-License-Identifier: Apache-2.0
| For details check: Apache-2.0_

.. _Apache-2.0: https://www.apache.org/licenses/LICENSE-2.0

.. </legal notes>  

*)
METHOD runCleanUp : CNM_ReturnTypes.SingleExecutionState
VAR_INPUT
	execute :BOOL;
	pause :BOOL;
END_VAR
END_METHOD

(*
## short summary
This method contains instructions and sequences for the ghost mode.
This mode is intended for running a machine without parts but with real device movements. Make sure to handle the missing part present signals.
If the node should do nothing, return a 'SUCCESS'.
It should run in an endless loop until the mode is stopped immedtiately or a stop request is raised (THIS^.modeControl.stopRequest).
This method is called automatically by the operation mode handler.

**attention**: If this method returns the state 'ERROR', the operation mode handler automatically disables the whole machine!

legal notes
=================
| SPDX-FileCopyrightText: © 2024 ekvip automation GmbH <info@ekvip.de>
| SPDX-License-Identifier: Apache-2.0
| For details check: Apache-2.0_

.. _Apache-2.0: https://www.apache.org/licenses/LICENSE-2.0

.. </legal notes>  

*)
METHOD runGhostMode : CNM_ReturnTypes.SingleExecutionState
VAR_INPUT
	execute :BOOL;
	pause :BOOL;
END_VAR
END_METHOD

(*
## short summary
This method contains instructions and sequences for the homing mode. It has to be overwritten for every node.
If the node should do nothing, return a 'SUCCESS'.
It should stop (return 'SUCCESS') if the node is in home state or a stop request is raised (THIS^.modeControl.stopRequest).
This method is called automatically by the operation mode handler.

**attention**: If this method returns the state 'ERROR', the operation mode handler automatically disables the whole machine!

legal notes
=================
| SPDX-FileCopyrightText: © 2024 ekvip automation GmbH <info@ekvip.de>
| SPDX-License-Identifier: Apache-2.0
| For details check: Apache-2.0_

.. _Apache-2.0: https://www.apache.org/licenses/LICENSE-2.0

.. </legal notes>  

*)
METHOD runHoming : CNM_ReturnTypes.SingleExecutionState
VAR_INPUT
	execute :BOOL;
	pause :BOOL;
END_VAR
END_METHOD

(*
## short summary
This method executes manual commands. It has to be overwritten for every node.
If the node should do nothing, return a 'SUCCESS'.
It should run endless until the manual mode is stopped via stop request or immediate stop.
This method is called automatically by the operation mode handler.

**attention**: If this method returns the state 'ERROR', the operation mode handler automatically disables the whole machine!

legal notes
=================
| SPDX-FileCopyrightText: © 2024 ekvip automation GmbH <info@ekvip.de>
| SPDX-License-Identifier: Apache-2.0
| For details check: Apache-2.0_

.. _Apache-2.0: https://www.apache.org/licenses/LICENSE-2.0

.. </legal notes>  

*)
METHOD runManual : CNM_ReturnTypes.SingleExecutionState
VAR_INPUT
	execute :BOOL;
	pause :BOOL;
END_VAR
END_METHOD

(*
## short summary
This method contains instructions and sequences for the referencing mode.
This mode is intended for referencing a machine with relative components, e.g. axes without absoulute position encodeing, torque driven axes (e.g. a press), coupling of master/slave axes.
If the node should do nothing, return a 'SUCCESS'.
It should run until all devices are referenced or the mode is stopped immedtiately or a stop request is raised (THIS^.modeControl.stopRequest).
This method is called automatically by the operation mode handler.

**attention**: If this method returns the state 'ERROR', the operation mode handler automatically disables the whole machine!

legal notes
=================
| SPDX-FileCopyrightText: © 2024 ekvip automation GmbH <info@ekvip.de>
| SPDX-License-Identifier: Apache-2.0
| For details check: Apache-2.0_

.. _Apache-2.0: https://www.apache.org/licenses/LICENSE-2.0

.. </legal notes>  

*)
METHOD runReferencing : CNM_ReturnTypes.SingleExecutionState
VAR_INPUT
	execute :BOOL;
	pause :BOOL;
END_VAR
END_METHOD

(*
## short summary
This method contains instructions and sequences for the service mode.
This mode is intended for supporting the maintanence of a machine, e.g. move components to a maintanence position, display and perform maintenance steps.
If the node should do nothing, return a 'SUCCESS'.
It should run until all servie requirements are done or the mode is stopped immedtiately or a stop request is raised (THIS^.modeControl.stopRequest).
This method is called automatically by the operation mode handler.

**attention**: If this method returns the state 'ERROR', the operation mode handler automatically disables the whole machine!

legal notes
=================
| SPDX-FileCopyrightText: © 2024 ekvip automation GmbH <info@ekvip.de>
| SPDX-License-Identifier: Apache-2.0
| For details check: Apache-2.0_

.. _Apache-2.0: https://www.apache.org/licenses/LICENSE-2.0

.. </legal notes>  

*)
METHOD runService : CNM_ReturnTypes.SingleExecutionState
VAR_INPUT
	execute :BOOL;
	pause :BOOL;
END_VAR
END_METHOD

(*
## short summary
This method simulates a node/unit/machine without physical movements, but with all data handling, e.g. handshakes between units, communication with production systems, loading of data.
This mode is intended for simulating the whole machine or single subunits by overwriting the mode for the subunit.
If the node should do nothing, return a 'SUCCESS'.
It should run endless until the mode is stopped immedtiately or a stop request is raised (THIS^.modeControl.stopRequest).
This method is called automatically by the operation mode handler.

**attention**: If this method returns the state 'ERROR', the operation mode handler automatically disables the whole machine!

legal notes
=================
| SPDX-FileCopyrightText: © 2024 ekvip automation GmbH <info@ekvip.de>
| SPDX-License-Identifier: Apache-2.0
| For details check: Apache-2.0_

.. _Apache-2.0: https://www.apache.org/licenses/LICENSE-2.0

.. </legal notes>  

*)
METHOD runSimulated : CNM_ReturnTypes.SingleExecutionState
VAR_INPUT
	execute :BOOL;
	pause :BOOL;
END_VAR
END_METHOD

END_INTERFACE

// ---- Project Information/F_GetCompany.TcPOU
// This function has been automatically generated from the project information.
{attribute 'signature_flag' := '1073741824'}
{attribute 'TcGenerated'}
{attribute 'no-analysis'}
FUNCTION F_GetCompany : WSTRING
VAR_INPUT
	
END_VAR

F_GetCompany := "ekvip automation GmbH";

END_FUNCTION

// ---- Project Information/F_GetTitle.TcPOU
// This function has been automatically generated from the project information.
{attribute 'signature_flag' := '1073741824'}
{attribute 'TcGenerated'}
{attribute 'no-analysis'}
FUNCTION F_GetTitle : WSTRING
VAR_INPUT
	
END_VAR

F_GetTitle := "CNM_OpModeHandlingInterfaces";

END_FUNCTION

// ---- Project Information/F_GetVersion.TcPOU
// This function has been automatically generated from the project information.
{attribute 'signature_flag' := '1073741824'}
{attribute 'TcGenerated'}
{attribute 'no-analysis'}
FUNCTION F_GetVersion : ST_LibVersion
VAR_INPUT
	
END_VAR

F_GetVersion.iMajor := 0;
F_GetVersion.iMinor := 1;
F_GetVersion.iBuild := 1;
F_GetVersion.iRevision := 0;
F_GetVersion.sVersion := '0.1.1.0';
F_GetVersion.nFlags := 0;

END_FUNCTION
